// TIA Portal V17 export
// export: Created 2021-12-03T08:13:14.2825263Z, ExportSetting WithDefaults, DisplayName Totally Integrated Automation Portal, DisplayVersion V17, DisplayName TIA Portal Openness, DisplayVersion V17, DisplayName TIA Portal Version Control Interface, DisplayVersion V17, DisplayName STEP 7 Professional, DisplayVersion V17, DisplayName STEP 7 Safety, DisplayVersion V17, DisplayName WinCC Advanced, DisplayVersion V17
FUNCTION "FFC_WriteOutputs" : Void   // FC60, F_FBD
VERSION : 0.1
// stored: AutoNumber false, IsIECCheckEnabled false, UDAEnableTagReadback false
BEGIN

REGION Network 1: 400 VAC Power Modulator NA2-1Q3
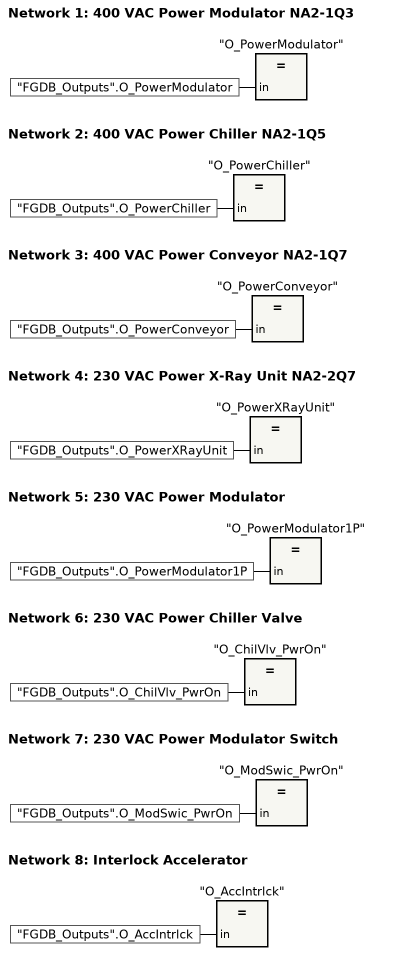
   "O_PowerModulator" := "FGDB_Outputs".O_PowerModulator;
END_REGION

REGION Network 2: 400 VAC Power Chiller NA2-1Q5
   "O_PowerChiller" := "FGDB_Outputs".O_PowerChiller;
END_REGION

REGION Network 3: 400 VAC Power Conveyor NA2-1Q7
   "O_PowerConveyor" := "FGDB_Outputs".O_PowerConveyor;
END_REGION

REGION Network 4: 230 VAC Power X-Ray Unit NA2-2Q7
   "O_PowerXRayUnit" := "FGDB_Outputs".O_PowerXRayUnit;
END_REGION

REGION Network 5: 230 VAC Power Modulator
   "O_PowerModulator1P" := "FGDB_Outputs".O_PowerModulator1P;
END_REGION

REGION Network 6: 230 VAC Power Chiller Valve
   "O_ChilVlv_PwrOn" := "FGDB_Outputs".O_ChilVlv_PwrOn;
END_REGION

REGION Network 7: 230 VAC Power Modulator Switch
   "O_ModSwic_PwrOn" := "FGDB_Outputs".O_ModSwic_PwrOn;
END_REGION

REGION Network 8: Interlock Accelerator
   "O_AccIntrlck" := "FGDB_Outputs".O_AccIntrlck;
END_REGION
END_FUNCTION
